// TwinCAT 3 PLC project testLibraryPrj
// ProgramVersion: 3.1.4024.0
// libraries:
//   Inputs and Outputs, * (MyCompany)
//   Tc2_Standard, * (Beckhoff Automation GmbH)
//   Tc2_System, * (Beckhoff Automation GmbH)
//   Tc3_Module, * (Beckhoff Automation GmbH)
// project tree:
//   / PlcTask.TcTTO
//   POUs/ MAIN.TcPOU

CONFIGURATION testLibraryPrj
    RESOURCE PLC ON TwinCAT3
        TASK PlcTask(INTERVAL := T#10ms, PRIORITY := 20);
        PROGRAM MAIN WITH PlcTask : MAIN;
    END_RESOURCE
END_CONFIGURATION

// ---- POUs/MAIN.TcPOU
PROGRAM MAIN
VAR
	numFactorial : ULINT;
	resFactorial : ULINT;
	setBool : BOOL;
END_VAR

IF setBool THEN
	resFactorial := IO.F_factorial(n := numFactorial);
	setBool := FALSE;	
END_IF

END_PROGRAM
